// TIA Portal V18 export
TYPE "UDT_BoilersOnOffSettings"
// stored: IsFailsafeCompliant false
   STRUCT
      OAT : Struct
         rBoiler1OATOff : Real := 18.0;
         rBoiler1OATOn : Real := 15.0;
         rBoiler2OAT1On : Real := 5.0;
         rBoiler2OAT1Off : Real := 10.0;
         rBoiler2OAT2On : Real := -5.0;
         rBoiler2OAT2Off : Real;
      END_STRUCT;
      PLCModeSelection : Struct
         cPreselectedOpModePLC : Byte;   // Вибор режиму роботи з PLC. 0-Вимкенено/1-Boiler1/2-Boiler2/3-B1+B2/4-Auto
         cActualOpModePLC : Byte;   // Актуальний режим роботи з PLC. 0-Вимкенено/1-Boiler1/2-Boiler2/3-B1+B2/4-Auto
      END_STRUCT;
   END_STRUCT;
END_TYPE
